Xinje XDPPro project, PLC1: XD3-32 (software 3.7.14 2021-12-24)

PROGRAM 梯形图

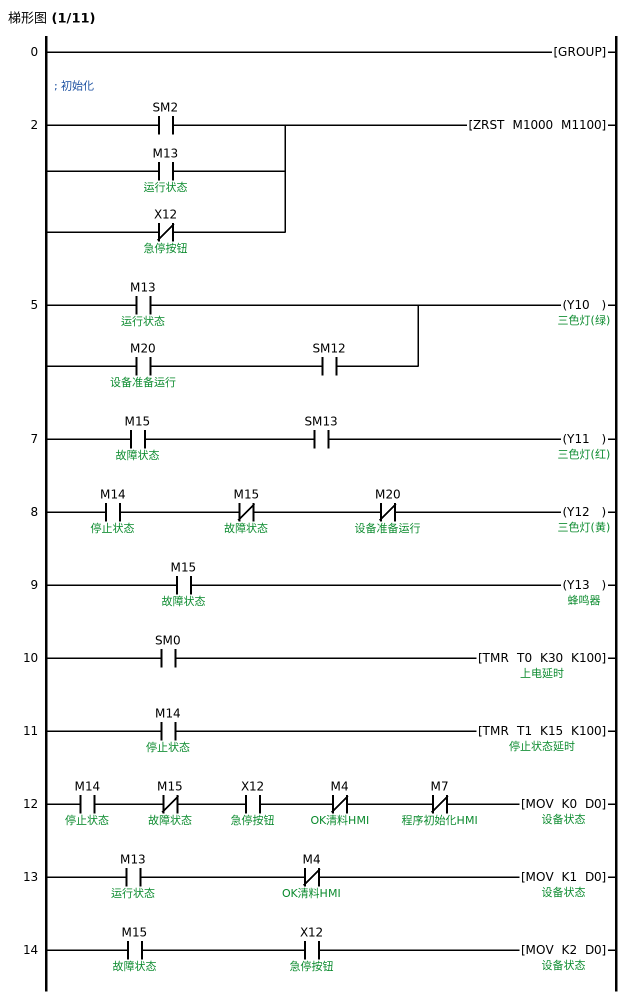
GROUP
; 初始化
LD     SM2
OR     M13	; 运行状态
ORI    X12	; 急停按钮
ZRST   M1000 M1100
LD     M13	; 运行状态
LD     M20	; 设备准备运行
AND    SM12
ORB
OUT    Y10	; 三色灯(绿)
LD     M15	; 故障状态
AND    SM13
OUT    Y11	; 三色灯(红)
LD     M14	; 停止状态
ANI    M15	; 故障状态
ANI    M20	; 设备准备运行
OUT    Y12	; 三色灯(黄)
LD     M15	; 故障状态
OUT    Y13	; 蜂鸣器
LD     SM0
TMR    T0 K30 K100	; 上电延时
LD     M14	; 停止状态
TMR    T1 K15 K100	; 停止状态延时
LD     M14	; 停止状态
ANI    M15	; 故障状态
AND    X12	; 急停按钮
ANI    M4	; OK清料HMI
ANI    M7	; 程序初始化HMI
MOV    K0 D0	; 设备状态
LD     M13	; 运行状态
ANI    M4	; OK清料HMI
MOV    K1 D0	; 设备状态
LD     M15	; 故障状态
AND    X12	; 急停按钮
MOV    K2 D0	; 设备状态

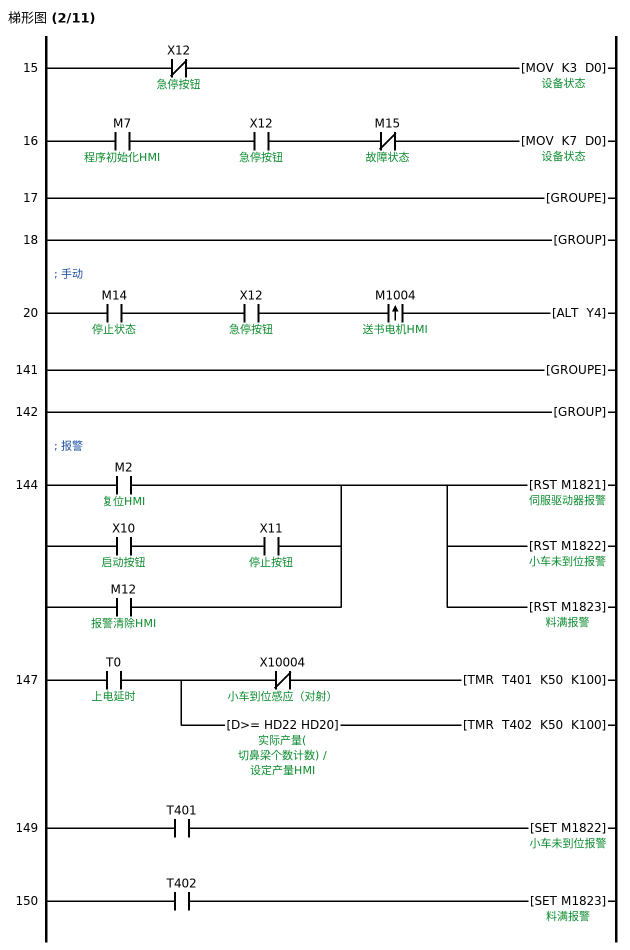
LDI    X12	; 急停按钮
MOV    K3 D0	; 设备状态
LD     M7	; 程序初始化HMI
AND    X12	; 急停按钮
ANI    M15	; 故障状态
MOV    K7 D0	; 设备状态
GROUPE
GROUP
; 手动
LD     M14	; 停止状态
AND    X12	; 急停按钮
ANDP   M1004	; 送书电机HMI
ALT    Y4
GROUPE
GROUP
; 报警
LD     M2	; 复位HMI
LD     X10	; 启动按钮
AND    X11	; 停止按钮
ORB
OR     M12	; 报警清除HMI
RST    M1821	; 伺服驱动器报警
RST    M1822	; 小车未到位报警
RST    M1823	; 料满报警
LD     T0	; 上电延时
MPS
ANI    X10004	; 小车到位感应（对射）
TMR    T401 K50 K100
MPP
DAND>= HD22 HD20	; 实际产量(切鼻梁个数计数) / 设定产量HMI
TMR    T402 K50 K100
LD     T401
SET    M1822	; 小车未到位报警
LD     T402
SET    M1823	; 料满报警

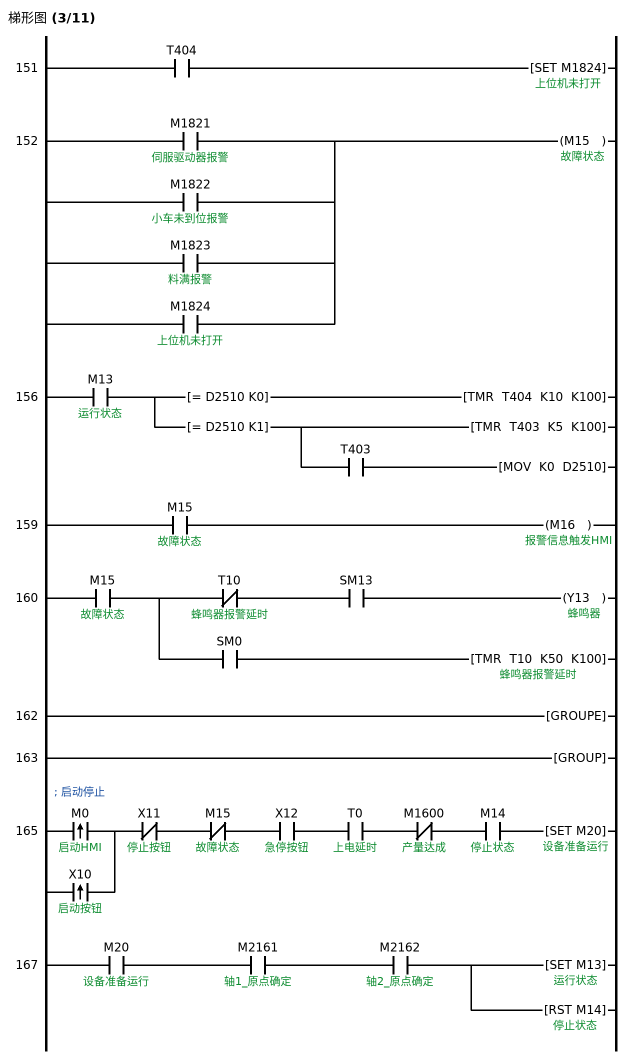
LD     T404
SET    M1824	; 上位机未打开
LD     M1821	; 伺服驱动器报警
OR     M1822	; 小车未到位报警
OR     M1823	; 料满报警
OR     M1824	; 上位机未打开
OUT    M15	; 故障状态
LD     M13	; 运行状态
MPS
AND=   D2510 K0
TMR    T404 K10 K100
MPP
AND=   D2510 K1
TMR    T403 K5 K100
AND    T403
MOV    K0 D2510
LD     M15	; 故障状态
OUT    M16	; 报警信息触发HMI
LD     M15	; 故障状态
MPS
ANI    T10	; 蜂鸣器报警延时
AND    SM13
OUT    Y13	; 蜂鸣器
MPP
AND    SM0
TMR    T10 K50 K100	; 蜂鸣器报警延时
GROUPE
GROUP
; 启动停止
LDP    M0	; 启动HMI
ORP    X10	; 启动按钮
ANI    X11	; 停止按钮
ANI    M15	; 故障状态
AND    X12	; 急停按钮
AND    T0	; 上电延时
ANI    M1600	; 产量达成
AND    M14	; 停止状态
SET    M20	; 设备准备运行
LD     M20	; 设备准备运行
AND    M2161	; 轴1_原点确定
AND    M2162	; 轴2_原点确定
SET    M13	; 运行状态
RST    M14	; 停止状态

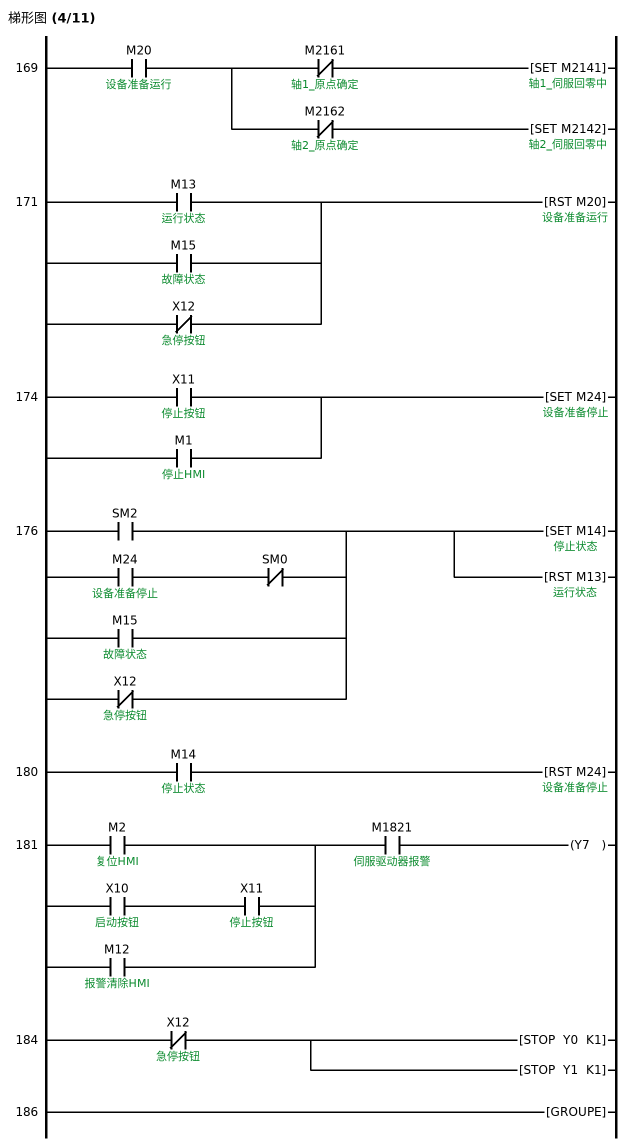
LD     M20	; 设备准备运行
MPS
ANI    M2161	; 轴1_原点确定
SET    M2141	; 轴1_伺服回零中
MPP
ANI    M2162	; 轴2_原点确定
SET    M2142	; 轴2_伺服回零中
LD     M13	; 运行状态
OR     M15	; 故障状态
ORI    X12	; 急停按钮
RST    M20	; 设备准备运行
LD     X11	; 停止按钮
OR     M1	; 停止HMI
SET    M24	; 设备准备停止
LD     SM2
LD     M24	; 设备准备停止
ANI    SM0
ORB
OR     M15	; 故障状态
ORI    X12	; 急停按钮
SET    M14	; 停止状态
RST    M13	; 运行状态
LD     M14	; 停止状态
RST    M24	; 设备准备停止
LD     M2	; 复位HMI
LD     X10	; 启动按钮
AND    X11	; 停止按钮
ORB
OR     M12	; 报警清除HMI
AND    M1821	; 伺服驱动器报警
OUT    Y7
LDI    X12	; 急停按钮
STOP   Y0 K1
STOP   Y1 K1
GROUPE

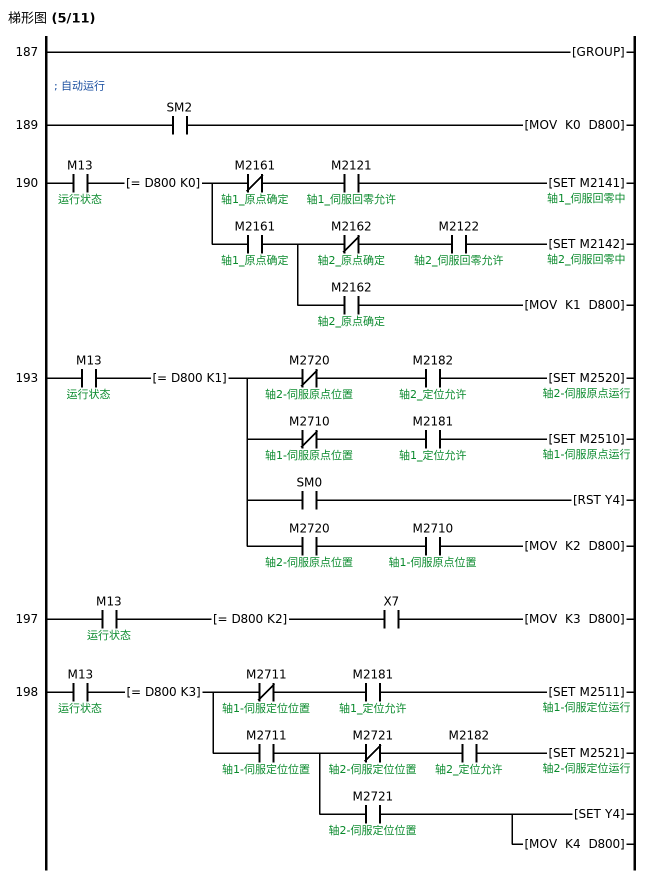
GROUP
; 自动运行
LD     SM2
MOV    K0 D800
LD     M13	; 运行状态
AND=   D800 K0
MPS
ANI    M2161	; 轴1_原点确定
AND    M2121	; 轴1_伺服回零允许
SET    M2141	; 轴1_伺服回零中
MPP
AND    M2161	; 轴1_原点确定
MPS
ANI    M2162	; 轴2_原点确定
AND    M2122	; 轴2_伺服回零允许
SET    M2142	; 轴2_伺服回零中
MPP
AND    M2162	; 轴2_原点确定
MOV    K1 D800
LD     M13	; 运行状态
AND=   D800 K1
MPS
ANI    M2720	; 轴2-伺服原点位置
AND    M2182	; 轴2_定位允许
SET    M2520	; 轴2-伺服原点运行
MRD
ANI    M2710	; 轴1-伺服原点位置
AND    M2181	; 轴1_定位允许
SET    M2510	; 轴1-伺服原点运行
MRD
AND    SM0
RST    Y4
MPP
AND    M2720	; 轴2-伺服原点位置
AND    M2710	; 轴1-伺服原点位置
MOV    K2 D800
LD     M13	; 运行状态
AND=   D800 K2
AND    X7
MOV    K3 D800
LD     M13	; 运行状态
AND=   D800 K3
MPS
ANI    M2711	; 轴1-伺服定位位置
AND    M2181	; 轴1_定位允许
SET    M2511	; 轴1-伺服定位运行
MPP
AND    M2711	; 轴1-伺服定位位置
MPS
ANI    M2721	; 轴2-伺服定位位置
AND    M2182	; 轴2_定位允许
SET    M2521	; 轴2-伺服定位运行
MPP
AND    M2721	; 轴2-伺服定位位置
SET    Y4
MOV    K4 D800

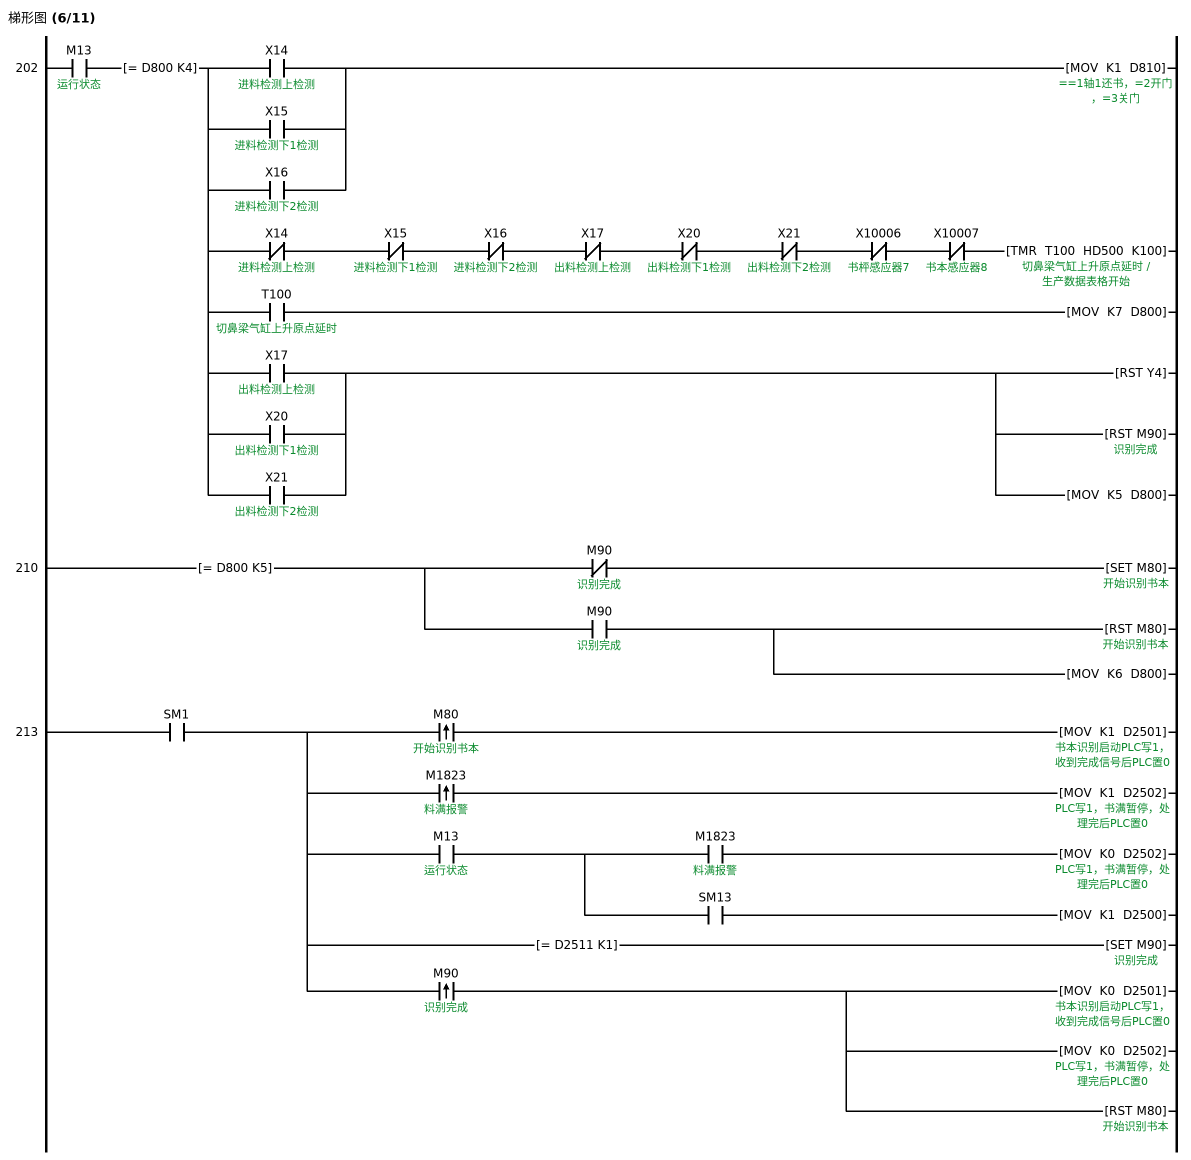
LD     M13	; 运行状态
AND=   D800 K4
MPS
LD     X14	; 进料检测上检测
OR     X15	; 进料检测下1检测
OR     X16	; 进料检测下2检测
ANB
MOV    K1 D810	; ==1轴1还书，=2开门，=3关门
MRD
ANI    X14	; 进料检测上检测
ANI    X15	; 进料检测下1检测
ANI    X16	; 进料检测下2检测
ANI    X17	; 出料检测上检测
ANI    X20	; 出料检测下1检测
ANI    X21	; 出料检测下2检测
ANI    X10006	; 书枰感应器7
ANI    X10007	; 书本感应器8
TMR    T100 HD500 K100	; 切鼻梁气缸上升原点延时 / 生产数据表格开始
MRD
AND    T100	; 切鼻梁气缸上升原点延时
MOV    K7 D800
MPP
LD     X17	; 出料检测上检测
OR     X20	; 出料检测下1检测
OR     X21	; 出料检测下2检测
ANB
RST    Y4
RST    M90	; 识别完成
MOV    K5 D800
LD=    D800 K5
MPS
ANI    M90	; 识别完成
SET    M80	; 开始识别书本
MPP
AND    M90	; 识别完成
RST    M80	; 开始识别书本
MOV    K6 D800
LD     SM1
MPS
ANDP   M80	; 开始识别书本
MOV    K1 D2501	; 书本识别启动PLC写1，收到完成信号后PLC置0
MRD
ANDP   M1823	; 料满报警
MOV    K1 D2502	; PLC写1，书满暂停，处理完后PLC置0
MRD
AND    M13	; 运行状态
MPS
AND    M1823	; 料满报警
MOV    K0 D2502	; PLC写1，书满暂停，处理完后PLC置0
MPP
AND    SM13
MOV    K1 D2500
MRD
AND=   D2511 K1
SET    M90	; 识别完成
MPP
ANDP   M90	; 识别完成
MOV    K0 D2501	; 书本识别启动PLC写1，收到完成信号后PLC置0
MOV    K0 D2502	; PLC写1，书满暂停，处理完后PLC置0
RST    M80	; 开始识别书本

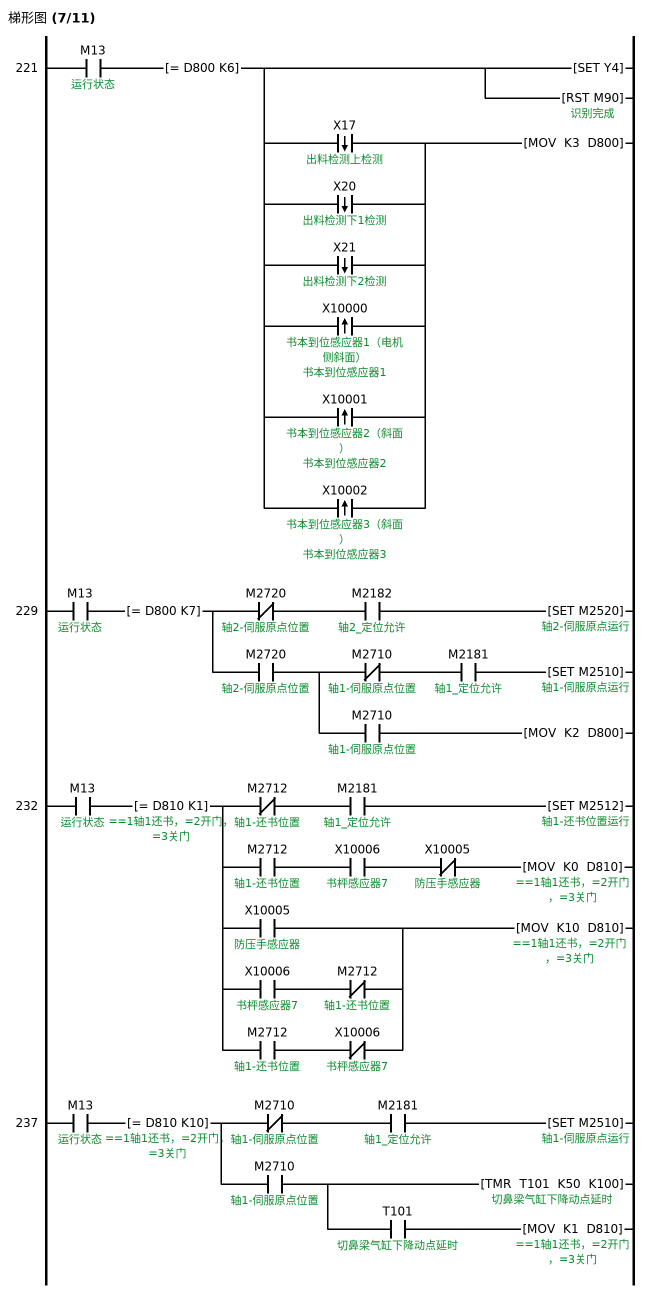
LD     M13	; 运行状态
AND=   D800 K6
SET    Y4
RST    M90	; 识别完成
LDF    X17	; 出料检测上检测
ORF    X20	; 出料检测下1检测
ORF    X21	; 出料检测下2检测
ORP    X10000	; 书本到位感应器1（电机侧斜面）       书本到位感应器1
ORP    X10001	; 书本到位感应器2（斜面）             书本到位感应器2
ORP    X10002	; 书本到位感应器3（斜面）             书本到位感应器3
ANB
MOV    K3 D800
LD     M13	; 运行状态
AND=   D800 K7
MPS
ANI    M2720	; 轴2-伺服原点位置
AND    M2182	; 轴2_定位允许
SET    M2520	; 轴2-伺服原点运行
MPP
AND    M2720	; 轴2-伺服原点位置
MPS
ANI    M2710	; 轴1-伺服原点位置
AND    M2181	; 轴1_定位允许
SET    M2510	; 轴1-伺服原点运行
MPP
AND    M2710	; 轴1-伺服原点位置
MOV    K2 D800
LD     M13	; 运行状态
AND=   D810 K1	; ==1轴1还书，=2开门，=3关门
MPS
ANI    M2712	; 轴1-还书位置
AND    M2181	; 轴1_定位允许
SET    M2512	; 轴1-还书位置运行
MRD
AND    M2712	; 轴1-还书位置
AND    X10006	; 书枰感应器7
ANI    X10005	; 防压手感应器
MOV    K0 D810	; ==1轴1还书，=2开门，=3关门
MPP
LD     X10005	; 防压手感应器
LD     X10006	; 书枰感应器7
ANI    M2712	; 轴1-还书位置
ORB
LD     M2712	; 轴1-还书位置
ANI    X10006	; 书枰感应器7
ORB
ANB
MOV    K10 D810	; ==1轴1还书，=2开门，=3关门
LD     M13	; 运行状态
AND=   D810 K10	; ==1轴1还书，=2开门，=3关门
MPS
ANI    M2710	; 轴1-伺服原点位置
AND    M2181	; 轴1_定位允许
SET    M2510	; 轴1-伺服原点运行
MPP
AND    M2710	; 轴1-伺服原点位置
TMR    T101 K50 K100	; 切鼻梁气缸下降动点延时
AND    T101	; 切鼻梁气缸下降动点延时
MOV    K1 D810	; ==1轴1还书，=2开门，=3关门

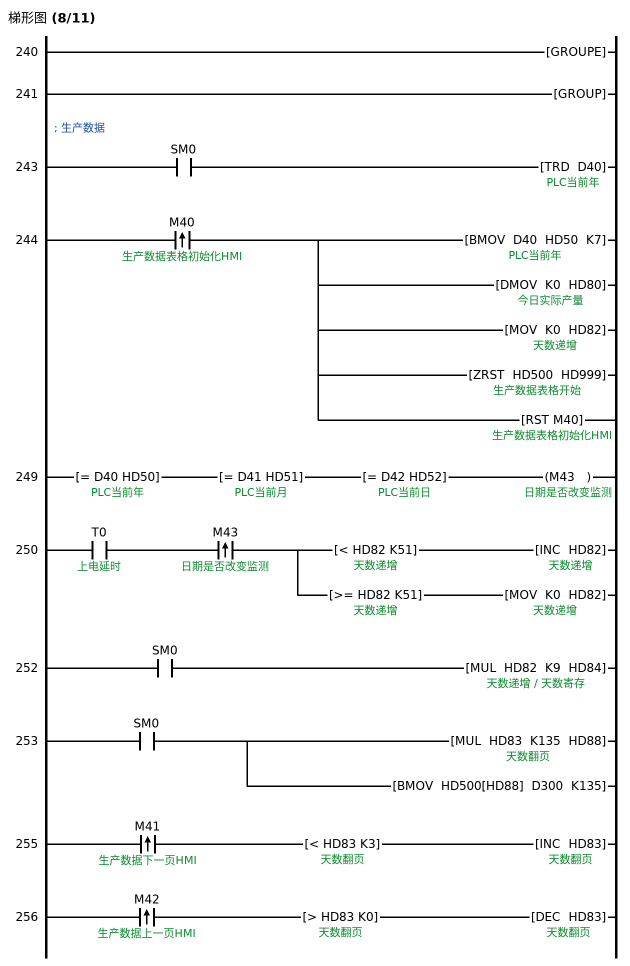
GROUPE
GROUP
; 生产数据
LD     SM0
TRD    D40	; PLC当前年
LDP    M40	; 生产数据表格初始化HMI
BMOV   D40 HD50 K7	; PLC当前年
DMOV   K0 HD80	; 今日实际产量
MOV    K0 HD82	; 天数递增
ZRST   HD500 HD999	; 生产数据表格开始
RST    M40	; 生产数据表格初始化HMI
LD=    D40 HD50	; PLC当前年
AND=   D41 HD51	; PLC当前月
AND=   D42 HD52	; PLC当前日
OUT    M43	; 日期是否改变监测
LD     T0	; 上电延时
ANDP   M43	; 日期是否改变监测
MPS
AND<   HD82 K51	; 天数递增
INC    HD82	; 天数递增
MPP
AND>=  HD82 K51	; 天数递增
MOV    K0 HD82	; 天数递增
LD     SM0
MUL    HD82 K9 HD84	; 天数递增 / 天数寄存
LD     SM0
MUL    HD83 K135 HD88	; 天数翻页
BMOV   HD500[HD88] D300 K135
LDP    M41	; 生产数据下一页HMI
AND<   HD83 K3	; 天数翻页
INC    HD83	; 天数翻页
LDP    M42	; 生产数据上一页HMI
AND>   HD83 K0	; 天数翻页
DEC    HD83	; 天数翻页

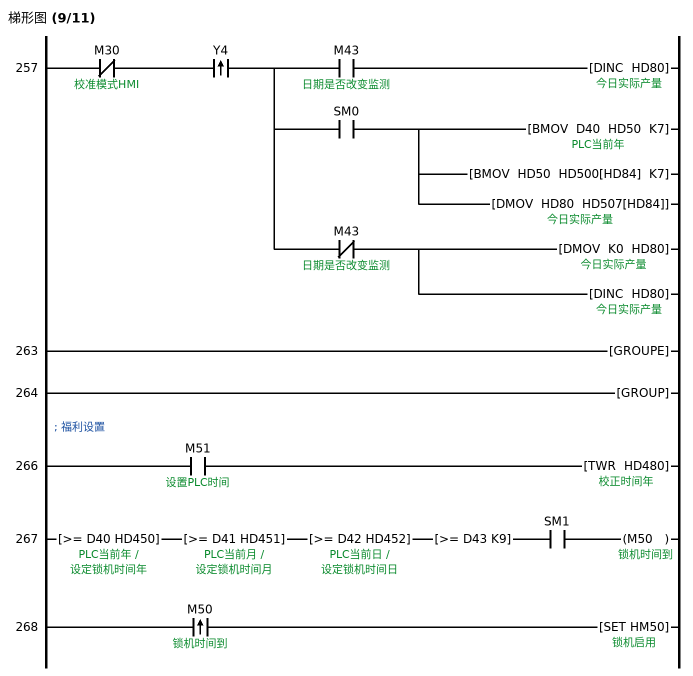
LDI    M30	; 校准模式HMI
ANDP   Y4
MPS
AND    M43	; 日期是否改变监测
DINC   HD80	; 今日实际产量
MRD
AND    SM0
BMOV   D40 HD50 K7	; PLC当前年
BMOV   HD50 HD500[HD84] K7
DMOV   HD80 HD507[HD84]	; 今日实际产量
MPP
ANI    M43	; 日期是否改变监测
DMOV   K0 HD80	; 今日实际产量
DINC   HD80	; 今日实际产量
GROUPE
GROUP
; 福利设置
LD     M51	; 设置PLC时间
TWR    HD480	; 校正时间年
LD>=   D40 HD450	; PLC当前年 / 设定锁机时间年
AND>=  D41 HD451	; PLC当前月 / 设定锁机时间月
AND>=  D42 HD452	; PLC当前日 / 设定锁机时间日
AND>=  D43 K9
AND    SM1
OUT    M50	; 锁机时间到
LDP    M50	; 锁机时间到
SET    HM50	; 锁机启用

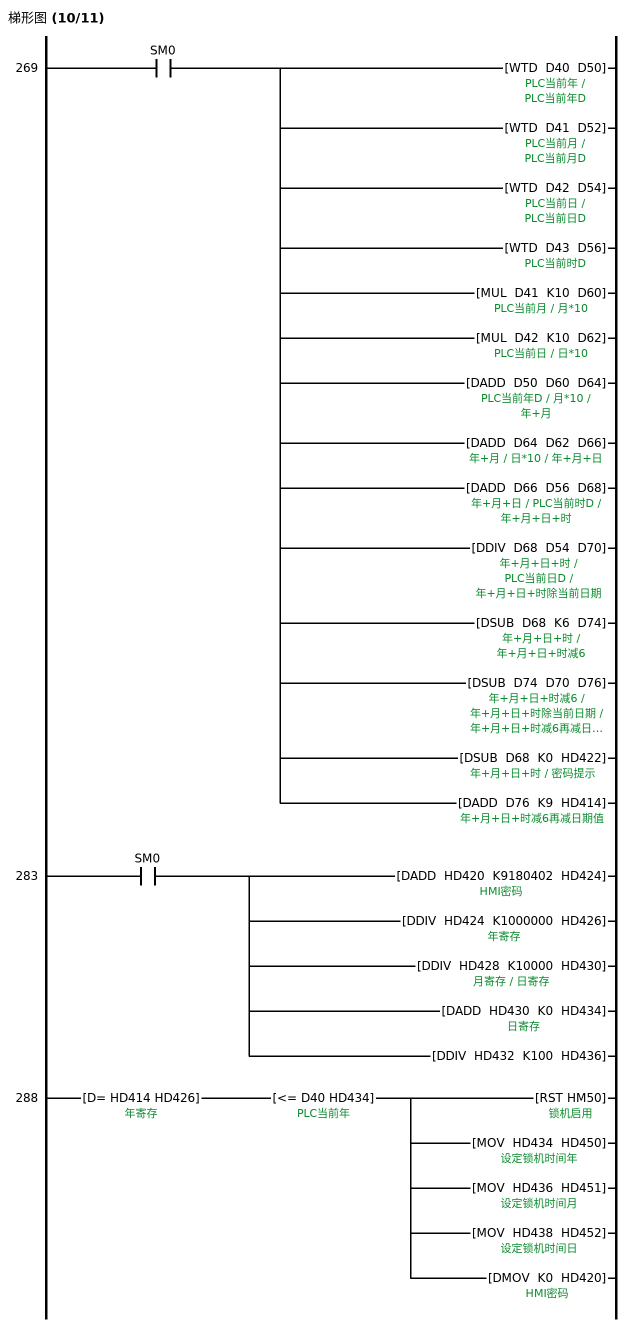
LD     SM0
WTD    D40 D50	; PLC当前年 / PLC当前年D
WTD    D41 D52	; PLC当前月 / PLC当前月D
WTD    D42 D54	; PLC当前日 / PLC当前日D
WTD    D43 D56	; PLC当前时D
MUL    D41 K10 D60	; PLC当前月 / 月*10
MUL    D42 K10 D62	; PLC当前日 / 日*10
DADD   D50 D60 D64	; PLC当前年D / 月*10 / 年+月
DADD   D64 D62 D66	; 年+月 / 日*10 / 年+月+日
DADD   D66 D56 D68	; 年+月+日 / PLC当前时D / 年+月+日+时
DDIV   D68 D54 D70	; 年+月+日+时 / PLC当前日D / 年+月+日+时除当前日期
DSUB   D68 K6 D74	; 年+月+日+时 / 年+月+日+时减6
DSUB   D74 D70 D76	; 年+月+日+时减6 / 年+月+日+时除当前日期 / 年+月+日+时减6再减日期值
DSUB   D68 K0 HD422	; 年+月+日+时 / 密码提示
DADD   D76 K9 HD414	; 年+月+日+时减6再减日期值
LD     SM0
DADD   HD420 K9180402 HD424	; HMI密码
DDIV   HD424 K1000000 HD426	; 年寄存
DDIV   HD428 K10000 HD430	; 月寄存 / 日寄存
DADD   HD430 K0 HD434	; 日寄存
DDIV   HD432 K100 HD436
DLD=   HD414 HD426	; 年寄存
AND<=  D40 HD434	; PLC当前年
RST    HM50	; 锁机启用
MOV    HD434 HD450	; 设定锁机时间年
MOV    HD436 HD451	; 设定锁机时间月
MOV    HD438 HD452	; 设定锁机时间日
DMOV   K0 HD420	; HMI密码

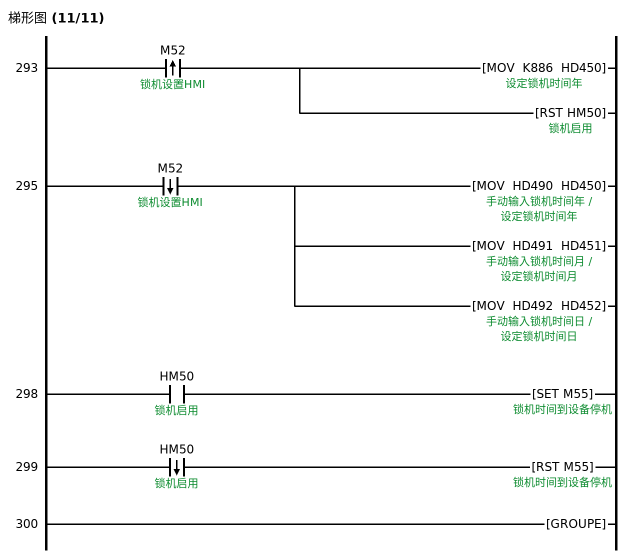
LDP    M52	; 锁机设置HMI
MOV    K886 HD450	; 设定锁机时间年
RST    HM50	; 锁机启用
LDF    M52	; 锁机设置HMI
MOV    HD490 HD450	; 手动输入锁机时间年 / 设定锁机时间年
MOV    HD491 HD451	; 手动输入锁机时间月 / 设定锁机时间月
MOV    HD492 HD452	; 手动输入锁机时间日 / 设定锁机时间日
LD     HM50	; 锁机启用
SET    M55	; 锁机时间到设备停机
LDF    HM50	; 锁机启用
RST    M55	; 锁机时间到设备停机
GROUPE

COMMENTS (devices not used above)
M3	急停HMI
M5	NG清料HMI
M6	轴复位HMI
M8	参数默认HMI
M9	产量清零HMI
M10	当前产量清零HMI
M21	軸总復位中
M22	设备复位中
M25	设备清料完成
M2042	轴2_JOG快慢速HMI
M2021	轴1_JOG- HMI
M2022	轴2_JOG- HMI
M2041	轴1_JOG快慢速HMI
M2002	轴2_JOG+ HMI
M1400	主送料伺服报警
M1401	送料鼻梁伺服报警
M1402	超声波报警
HD200	轴2_JOG快速度HMI
HD202	轴2_JOG慢速度HMI
HD204	轴2_JOG速度寄存
HD206	轴2_JOG增量
HD208	轴2_JOG位置寄存
HD210	轴2_回零速度
HD212	轴2_运行速度HMI
HD214	轴2_自动加速度
HD215	轴2_自动减速度
HD218	轴2_定位位置寄存
D2100	轴1_JOG快速度
D2102	轴1_JOG慢速度
D2104	轴1_JOG速度寄存
D2106	轴1_JOG增量
D2108	轴1_JOG位置寄存
D2110	轴1_回零速度
D2112	轴1_运行速度
D2114	轴1_自动加速度
D2115	轴1_自动减速度
D2116	轴1_JOG加速度
D2117	轴1_JOG减速度
D2118	轴1_定位位置寄存
HD216	轴2_手动加速度
HD217	轴2_手动减速度
M1200	快慢速切换HMI
Y15	进料输送皮带（KA2)
HD8	切鼻梁个数计数
HD220	轴2_鼻梁长度设置HMI
HD12	滚刀切料个数计数
M2001	轴1_JOG+ HMI
HD40	Y0当前脉冲值记忆
HD42	Y1当前脉冲值记忆
T2	超声波休眠延时
HD2	超声波休眠时间
T3	超声运行延时
HD300	生产速度HMI
HD310	鼻梁滚轮周长HMI
HD100	轴1_JOG快速度HMI
HD102	轴1_JOG慢速度HMI
HD104	轴1_JOG速度寄存
HD106	轴1_JOG增量
HD108	轴1_JOG位置寄存
HD110	轴1_回零速度
HD112	轴1_运行速度HMI
HD114	轴1_自动加速度
HD115	轴1_自动减速度
HD116	轴1_JOG加速度
HD117	轴1_JOG减速度
HD118	轴1_定位位置寄存
D108	鼻梁长度计算脉冲结果
D100	K750浮点数
D104	鼻梁长度计算脉冲结果寄存
D142	输出脉冲频率浮点数
HD32	生产效率寄存2
HD30	生产效率寄存1
HM30	内置鼻梁标志/外置鼻梁HMI
HD24	滚刀切料个数计数
HD34	生产效率
HM32	校准完成
M1403	设备未校准
M107	主轴清零标志
M102	送鼻梁运行开始
HM3	急停后切断鼻梁
M1404	急停后手动切断鼻梁再启动！
M18	手动操作记忆标志
HD507	当日实际产量
HD400	当前时间年
HD401	当前时间月
HD402	当前时间日
HD403	当前时间时
HD453	设定锁机时间时
HD481	校正时间月
HD482	校正时间日
HD483	校正时间时
D72	年+月+日+时除当前日期得商
HD28	累计产量
X10003	小车感应光栅
M2101	轴1_伺服回零HMI
M2102	轴2_伺服回零HMI
M2201	轴1_JOG连续/增量HMI
M2202	轴2_JOG连续/增量HMI
M2241	轴1_增量JOG运行
M2242	轴2_增量JOG运行
M2310	轴1-伺服原点运行HMI
M2311	轴1-伺服定位运行HMI
M2320	轴2-伺服原点运行HMI
M2321	轴2-伺服定位运行HMI
HD894	轴1_设置每次回零计数HMI
HD895	轴1_当前每次回零计数
HD900	轴2_JOG快速度HMI
HD902	轴2_JOG慢速度HMI
HD904	轴2_JOG速度寄存
HD906	轴2_JOG增量
HD908	轴2_JOG位置寄存
HD910	轴2_回零速度
HD912	轴2_运行速度HMI
HD914	轴2_自动加速度
HD915	轴2_自动减速度
HD916	轴2_手动加速度
HD917	轴2_手动减速度
HD918	轴2_定位位置寄存
HD920	轴2__原点位置HMI
HD922	轴2__定位位置HMI
HD994	轴2_设置每次回零计数HMI
HD995	轴2_当前每次回零计数
HD800	轴1_JOG快速度HMI
HD802	轴1_JOG慢速度HMI
HD804	轴1_JOG速度寄存
HD806	轴1_JOG增量
HD808	轴1_JOG位置寄存
HD810	轴1_回零速度
HD812	轴1_运行速度HMI
HD814	轴1_自动加速度
HD815	轴1_自动减速度
HD816	轴1_JOG加速度
HD817	轴1_JOG减速度
HD818	轴1_定位位置寄存
HD820	轴1__原点位置HMI
HD822	轴1__定位位置HMI
D851	轴1-回原点流程
HD890	轴1-正软限位HMI
HD892	轴1-负软限位HMI
T422	轴1 启动
HD888	轴1—当前脉冲数
HD988	轴2当前脉冲数
M1006	使能HMI
D852	轴2-回原流程
T424	轴2定位允许
M2312	还书位置运行-HMI